(* Logix 5000 project; controller Joltek_RA_5069PLC002 vendor 1 type 14 code 226 rev 34.15; software revision 34.04; part 3 of 3 *)

PROGRAM SafetyProgram   (* main routine MainRoutine, safety *)

ROUTINE MainRoutine   (* ladder *)
END_ROUTINE
END_PROGRAM
